FUNCTION_BLOCK JackPlaceWP (* Basic Function Block Type *)
  (* Standard: 61499-2 *)
  (* Version 0.0, 9/26/2018, dmidro, nxtControl GmbH, Template *)
  PACKAGE Main;
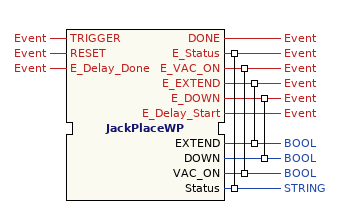
  EVENT_INPUT
    TRIGGER; (* Normal Execution Request *)
    RESET;
    E_Delay_Done;
  END_EVENT
  EVENT_OUTPUT
    DONE; (* Initialization Confirm *)
    E_Status WITH Status;
    E_VAC_ON WITH VAC_ON;
    E_EXTEND WITH EXTEND;
    E_DOWN WITH DOWN;
    E_Delay_Start;
  END_EVENT
  VAR_OUTPUT
    EXTEND : BOOL;
    DOWN : BOOL;
    VAC_ON : BOOL;
    Status : STRING;
  END_VAR
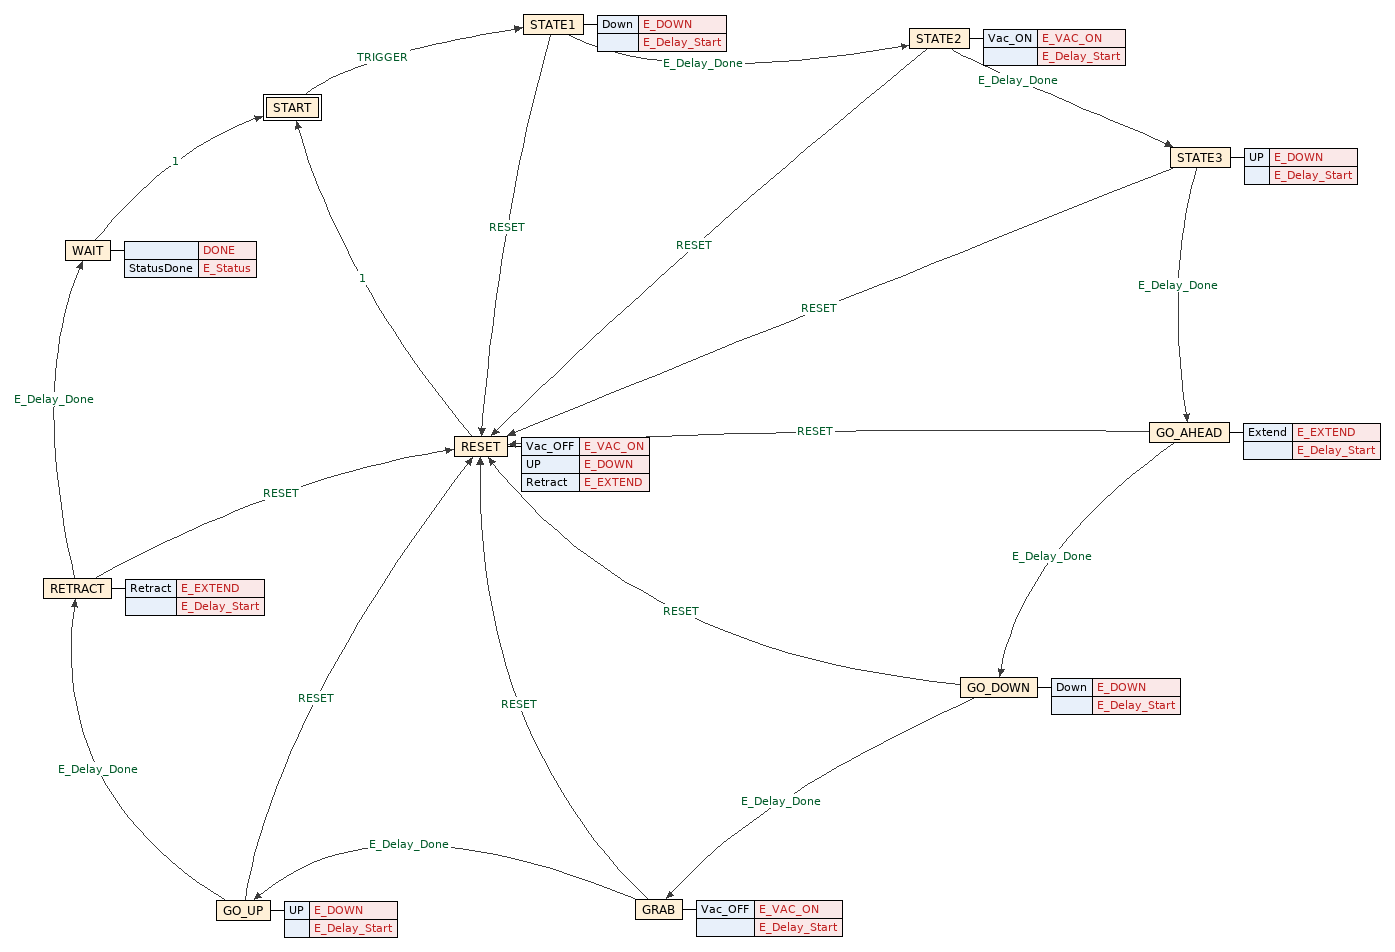
  EC_STATES
    START; (* Initial State *)
    GO_AHEAD : Extend -> E_EXTEND, -> E_Delay_Start;
    GO_DOWN : Down -> E_DOWN, -> E_Delay_Start;
    GRAB : Vac_OFF -> E_VAC_ON, -> E_Delay_Start;
    GO_UP : UP -> E_DOWN, -> E_Delay_Start;
    RETRACT : Retract -> E_EXTEND, -> E_Delay_Start;
    RESET : Vac_OFF -> E_VAC_ON, UP -> E_DOWN, Retract -> E_EXTEND;
    WAIT : -> DONE, StatusDone -> E_Status;
    STATE1 : Down -> E_DOWN, -> E_Delay_Start;
    STATE2 : Vac_ON -> E_VAC_ON, -> E_Delay_Start;
    STATE3 : UP -> E_DOWN, -> E_Delay_Start;
  END_STATES
  EC_TRANSITIONS
    START TO STATE1 := TRIGGER;
    GO_AHEAD TO GO_DOWN := E_Delay_Done;
    GO_DOWN TO GRAB := E_Delay_Done;
    GRAB TO GO_UP := E_Delay_Done;
    GO_UP TO RETRACT := E_Delay_Done;
    RETRACT TO WAIT := E_Delay_Done;
    WAIT TO START := 1;
    GO_AHEAD TO RESET := RESET;
    GO_DOWN TO RESET := RESET;
    GRAB TO RESET := RESET;
    GO_UP TO RESET := RESET;
    RETRACT TO RESET := RESET;
    RESET TO START := 1;
    STATE1 TO STATE2 := E_Delay_Done;
    STATE2 TO STATE3 := E_Delay_Done;
    STATE1 TO RESET := RESET;
    STATE2 TO RESET := RESET;
    STATE3 TO GO_AHEAD := E_Delay_Done;
    STATE3 TO RESET := RESET;
  END_TRANSITIONS
  ALGORITHM Down IN ST:
DOWN := TRUE;
E_Delay_Done := FALSE;
  END_ALGORITHM
  ALGORITHM Vac_ON IN ST:
VAC_ON := TRUE;
E_Delay_Done := FALSE;
  END_ALGORITHM
  ALGORITHM UP IN ST:
DOWN := FALSE;
E_Delay_Done := FALSE;
  END_ALGORITHM
  ALGORITHM Extend IN ST:
EXTEND := TRUE ;
E_Delay_Done := FALSE;
  END_ALGORITHM
  ALGORITHM Vac_OFF IN ST:
VAC_ON := FALSE ;
E_Delay_Done := FALSE;
  END_ALGORITHM
  ALGORITHM Retract IN ST:
EXTEND := FALSE ;
E_Delay_Done := FALSE;
  END_ALGORITHM
  ALGORITHM StatusStarted IN ST:
Status := 'S';
E_Delay_Done := FALSE;
  END_ALGORITHM
  ALGORITHM StatusDone IN ST:
Status := 'PLACE_D';
E_Delay_Done := FALSE;
  END_ALGORITHM
END_FUNCTION_BLOCK
